// Mitsubishi GX Works2 project: star-delta connection circuit   PLC: FX1N/FX1NC

PROGRAM MAIN
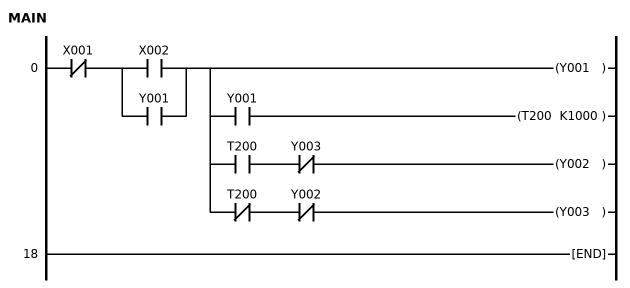
0     LDI     X001
      LD      X002
      OR      Y001
      ANB
      OUT     Y001
      MPS
      AND     Y001
      OUT     T200 K1000
      MRD
      AND     T200
      ANI     Y003
      OUT     Y002
      MPP
      ANI     T200
      ANI     Y002
      OUT     Y003
18    END
END_PROGRAM
